(* Logix 5000 project; controller Turck_IOLink_All_Full_AOIs_V0_1 vendor 1 type 14 code 176 rev 32.11; software revision 32.00; part 4 of 7 *)
(* tags used below, declared in another part *)
   Port : INT;
   Common_Data : Turck_IOLink_Common_Data;   // Controller Tag of Process Data
   Units : SINT;   // Index 0x54 Subindex 1 - Change the Displayed Unit 0 = bar 1 = psi 2 = kPa 3 = MPa 4-14 = See Manual
   Rotate_Display : SINT;   // Index 0x5B - Subindex 1 - Display Rotation 0 = 0degrees 1 = 180 degrees
   Error : BOOL;
   Done : DINT;
   Error_DINT : DINT;
   Pending : DINT;
   Pending_or_Active : DINT;
   Units_Prev : SINT;
   StartupDone : BOOL;
   Active : DINT;
   Read_ONS : DINT;
   MyTicketNum : INT[32];
   Write : DINT;
   Write_ONS : DINT;
   WriteRequest : DINT;
   DoneCount : DINT;
   Status : DINT;
   ErrorCount : DINT;
   ReadRequest : DINT;
   Rotate_Display_Prev : SINT;
   Process_Data_Profile : SINT;
   Max_Pressure_Recorded_Raw : INT;
   Every_Min_Poll_TON : TIMER;
   Min_Recorded_Pressure_Raw : INT;
(* Turck_PS510_10V_Full, continued *)

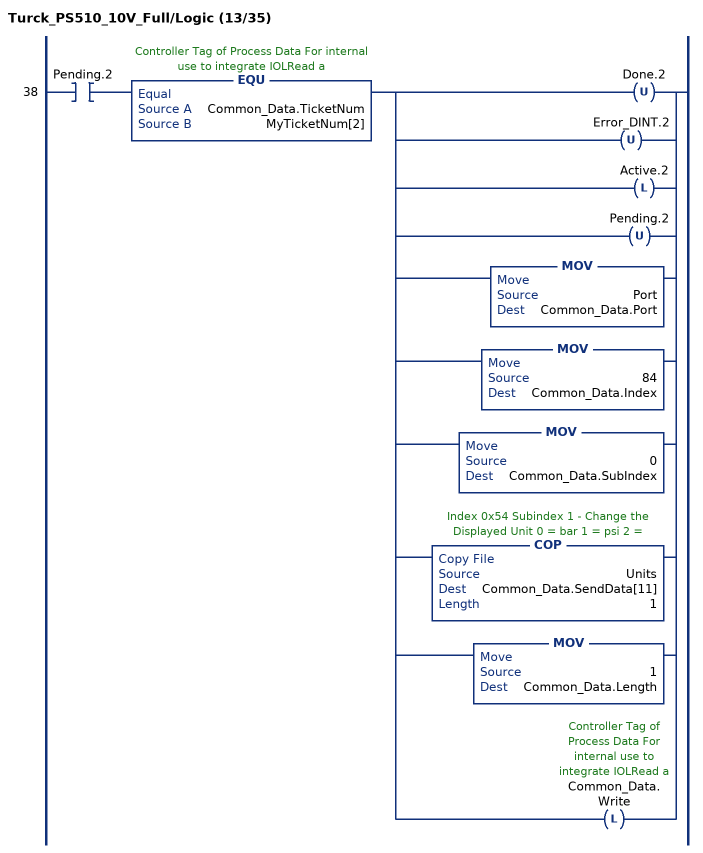
   [picture p75: Turck_PS510_10V_Full/Logic rungs 38-38]
   38: XIC(Pending.2)EQU(Common_Data.TicketNum,MyTicketNum[2])[OTU(Done.2) ,OTU(Error_DINT.2) ,OTL(Active.2) ,OTU(Pending.2) ,MOV(Port,Common_Data.Port) ,MOV(84,Common_Data.Index) ,MOV(0,Common_Data.SubIndex) ,COP(Units,Common_Data.SendData[11],1) ,MOV(1,Common_Data.Length) ,OTL(Common_Data.Write) ];
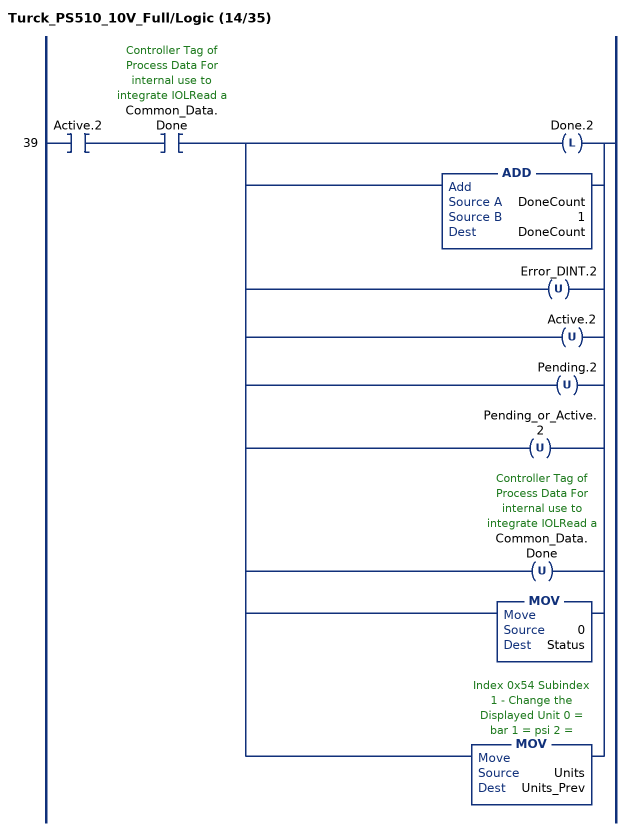
   39: XIC(Active.2)XIC(Common_Data.Done)[OTL(Done.2) ,ADD(DoneCount,1,DoneCount) ,OTU(Error_DINT.2) ,OTU(Active.2) ,OTU(Pending.2) ,OTU(Pending_or_Active.2) ,OTU(Common_Data.Done) ,MOV(0,Status) ,MOV(Units,Units_Prev) ];
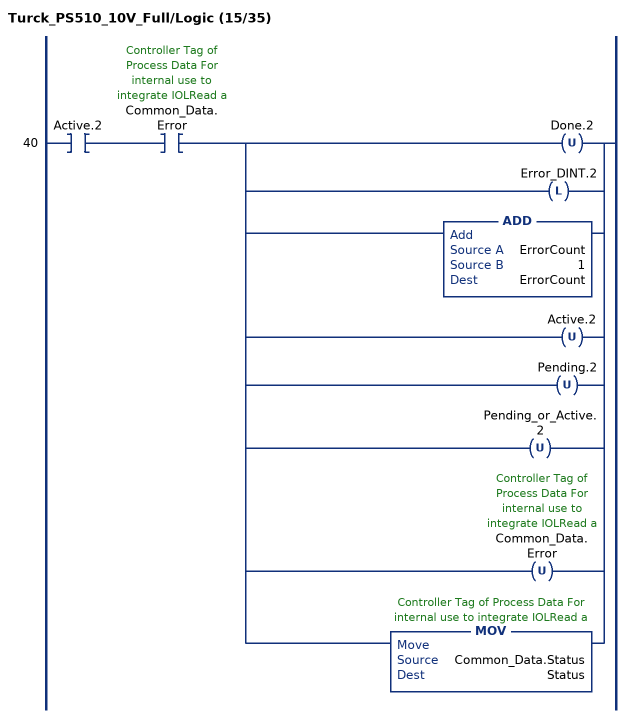
   40: XIC(Active.2)XIC(Common_Data.Error)[OTU(Done.2) ,OTL(Error_DINT.2) ,ADD(ErrorCount,1,ErrorCount) ,OTU(Active.2) ,OTU(Pending.2) ,OTU(Pending_or_Active.2) ,OTU(Common_Data.Error) ,MOV(Common_Data.Status,Status) ];
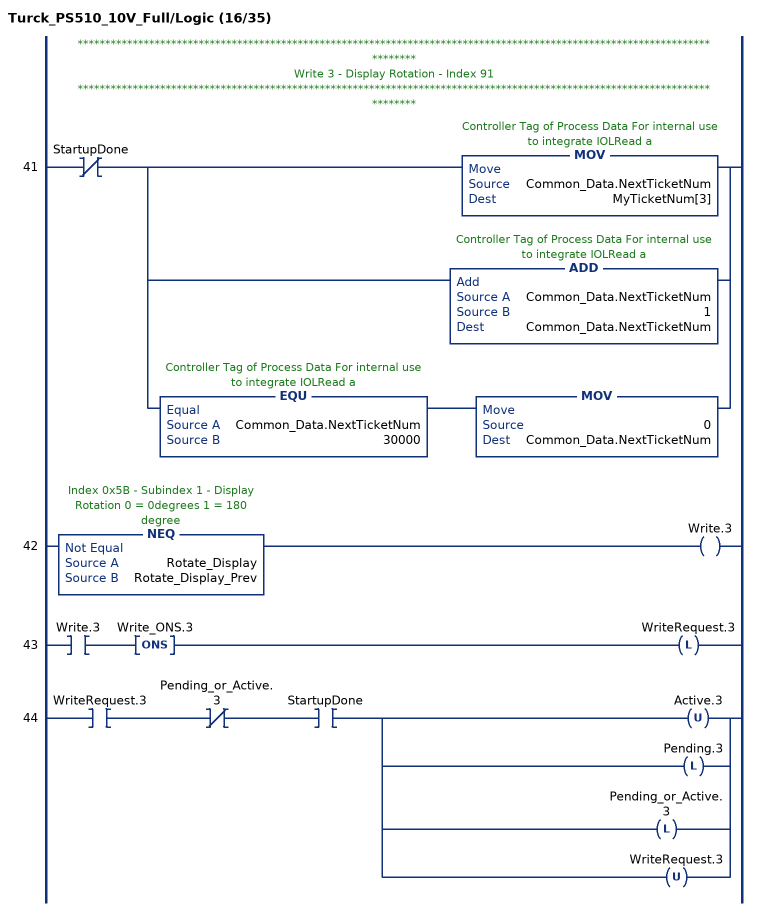
   // ***************************************************************************************************************************
   // Write 3 - Display Rotation - Index 91
   // ***************************************************************************************************************************
   41: XIO(StartupDone)[MOV(Common_Data.NextTicketNum,MyTicketNum[3]) ,ADD(Common_Data.NextTicketNum,1,Common_Data.NextTicketNum) ,EQU(Common_Data.NextTicketNum,30000) MOV(0,Common_Data.NextTicketNum) ];
   42: NEQ(Rotate_Display,Rotate_Display_Prev)OTE(Write.3);
   43: XIC(Write.3)ONS(Write_ONS.3)OTL(WriteRequest.3);
   44: XIC(WriteRequest.3)XIO(Pending_or_Active.3)XIC(StartupDone)[OTU(Active.3) ,OTL(Pending.3) ,OTL(Pending_or_Active.3) ,OTU(WriteRequest.3) ];
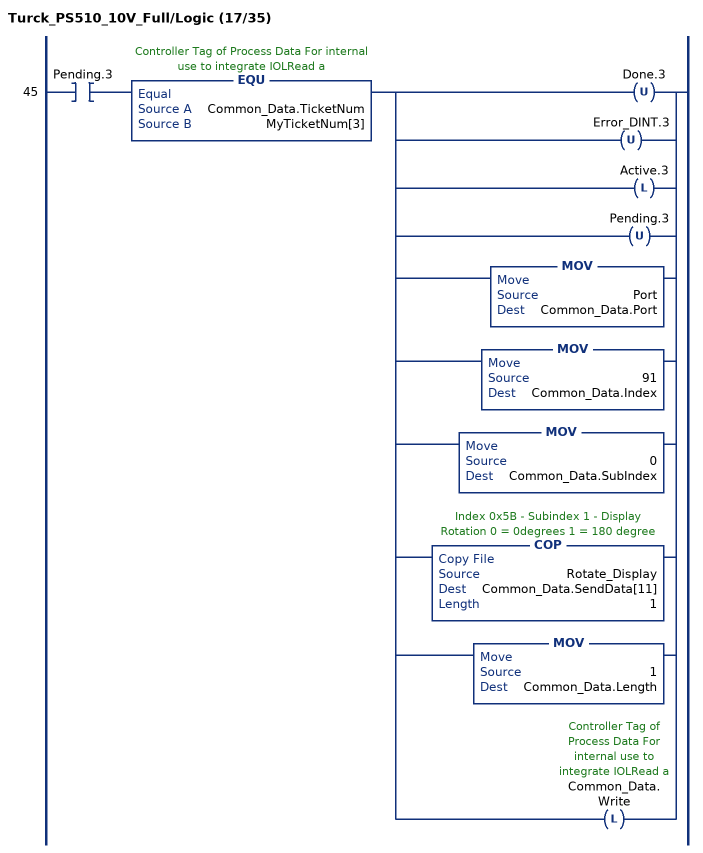
   45: XIC(Pending.3)EQU(Common_Data.TicketNum,MyTicketNum[3])[OTU(Done.3) ,OTU(Error_DINT.3) ,OTL(Active.3) ,OTU(Pending.3) ,MOV(Port,Common_Data.Port) ,MOV(91,Common_Data.Index) ,MOV(0,Common_Data.SubIndex) ,COP(Rotate_Display,Common_Data.SendData[11],1) ,MOV(1,Common_Data.Length) ,OTL(Common_Data.Write) ];
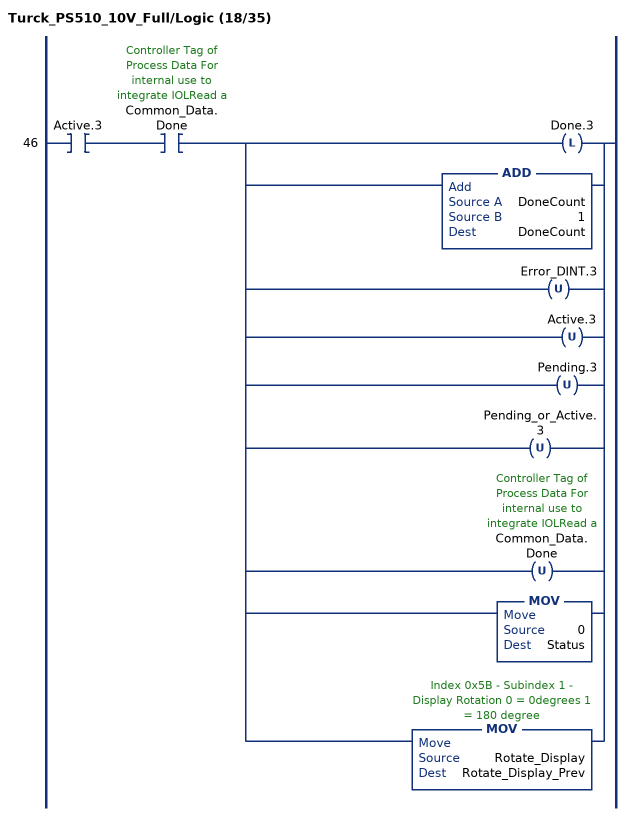
   46: XIC(Active.3)XIC(Common_Data.Done)[OTL(Done.3) ,ADD(DoneCount,1,DoneCount) ,OTU(Error_DINT.3) ,OTU(Active.3) ,OTU(Pending.3) ,OTU(Pending_or_Active.3) ,OTU(Common_Data.Done) ,MOV(0,Status) ,MOV(Rotate_Display,Rotate_Display_Prev) ];
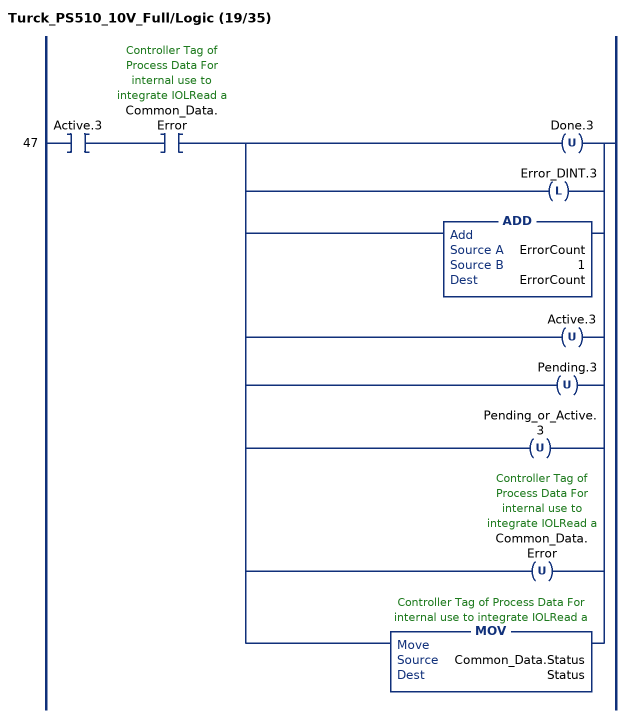
   47: XIC(Active.3)XIC(Common_Data.Error)[OTU(Done.3) ,OTL(Error_DINT.3) ,ADD(ErrorCount,1,ErrorCount) ,OTU(Active.3) ,OTU(Pending.3) ,OTU(Pending_or_Active.3) ,OTU(Common_Data.Error) ,MOV(Common_Data.Status,Status) ];
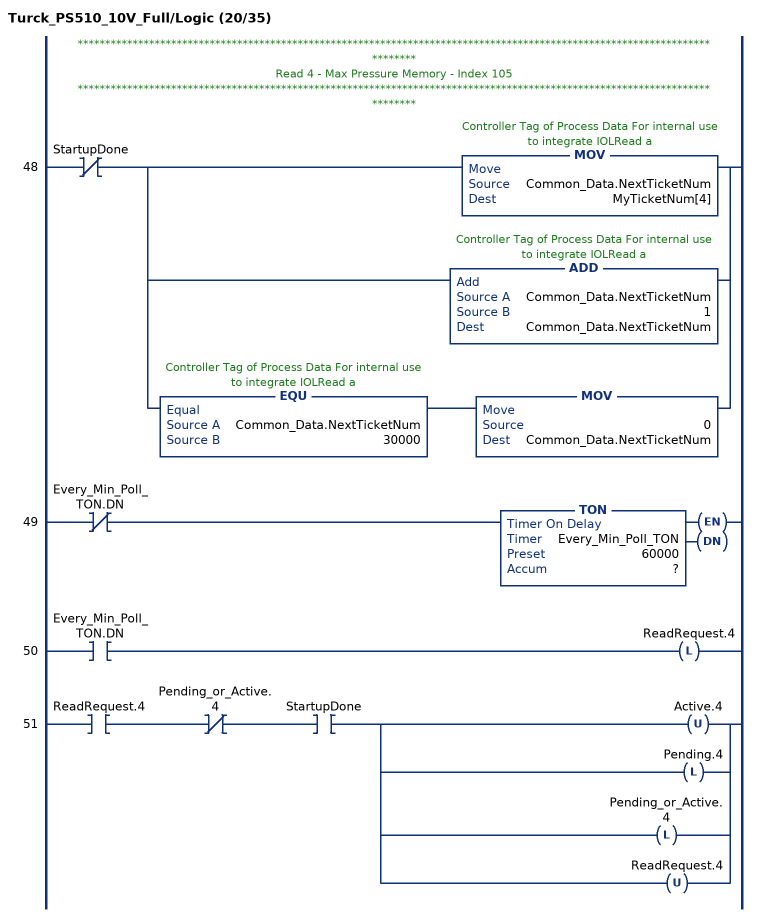
   // ***************************************************************************************************************************
   // Read 4 - Max Pressure Memory - Index 105
   // ***************************************************************************************************************************
   48: XIO(StartupDone)[MOV(Common_Data.NextTicketNum,MyTicketNum[4]) ,ADD(Common_Data.NextTicketNum,1,Common_Data.NextTicketNum) ,EQU(Common_Data.NextTicketNum,30000) MOV(0,Common_Data.NextTicketNum) ];
   49: XIO(Every_Min_Poll_TON.DN)TON(Every_Min_Poll_TON,?,?);
   50: XIC(Every_Min_Poll_TON.DN)OTL(ReadRequest.4);
   51: XIC(ReadRequest.4)XIO(Pending_or_Active.4)XIC(StartupDone)[OTU(Active.4) ,OTL(Pending.4) ,OTL(Pending_or_Active.4) ,OTU(ReadRequest.4) ];
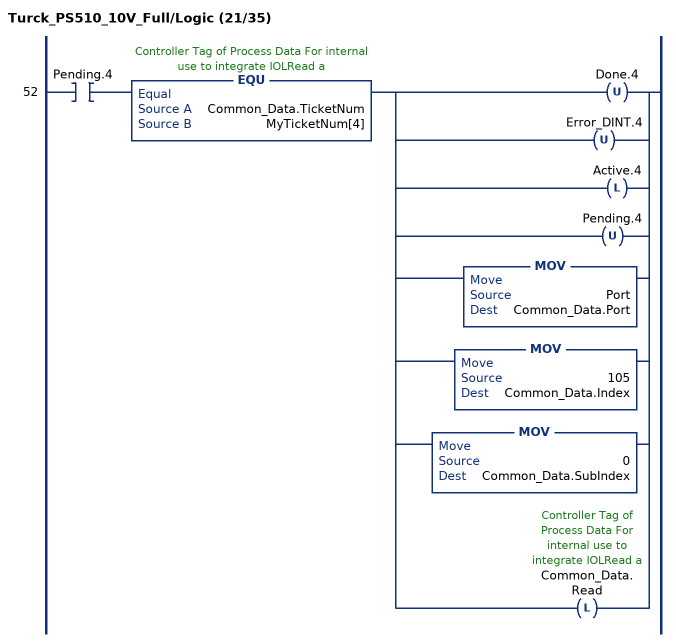
   52: XIC(Pending.4)EQU(Common_Data.TicketNum,MyTicketNum[4])[OTU(Done.4) ,OTU(Error_DINT.4) ,OTL(Active.4) ,OTU(Pending.4) ,MOV(Port,Common_Data.Port) ,MOV(105,Common_Data.Index) ,MOV(0,Common_Data.SubIndex) ,OTL(Common_Data.Read) ];
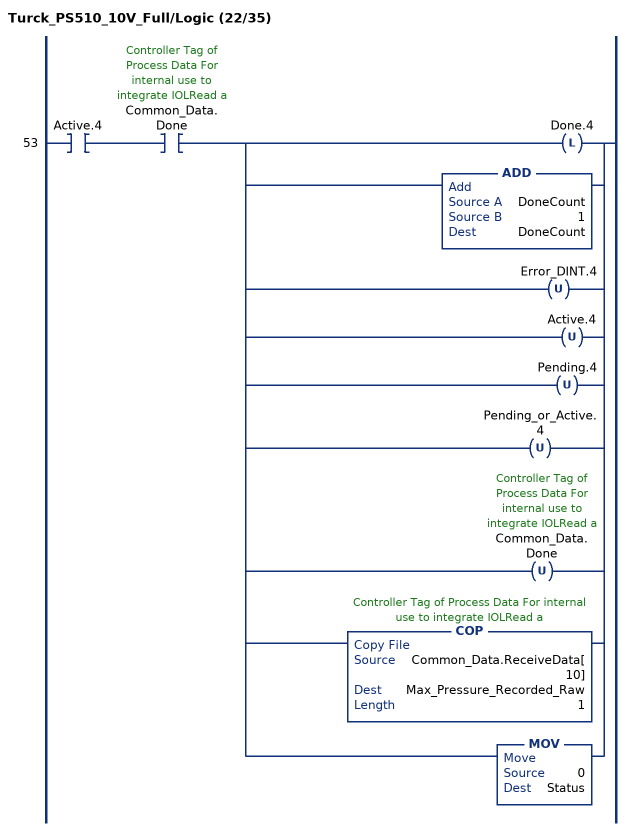
   53: XIC(Active.4)XIC(Common_Data.Done)[OTL(Done.4) ,ADD(DoneCount,1,DoneCount) ,OTU(Error_DINT.4) ,OTU(Active.4) ,OTU(Pending.4) ,OTU(Pending_or_Active.4) ,OTU(Common_Data.Done) ,COP(Common_Data.ReceiveData[10],Max_Pressure_Recorded_Raw,1) ,MOV(0,Status) ];
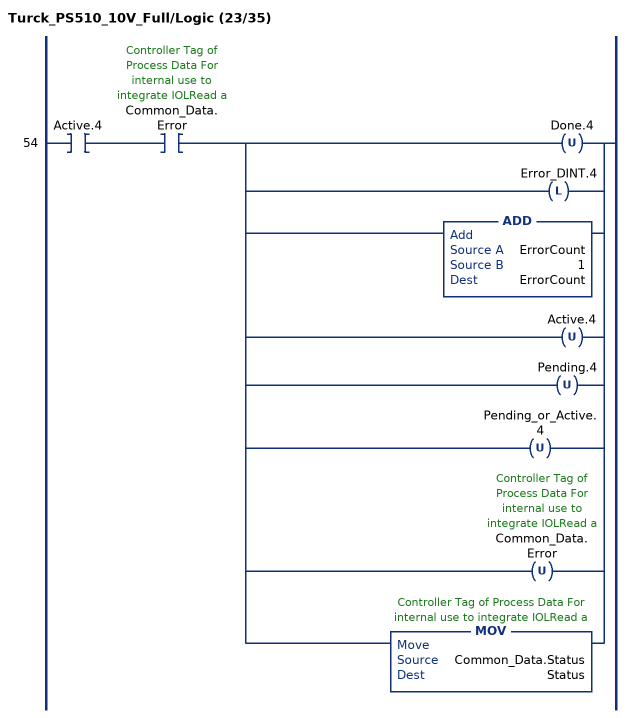
   54: XIC(Active.4)XIC(Common_Data.Error)[OTU(Done.4) ,OTL(Error_DINT.4) ,ADD(ErrorCount,1,ErrorCount) ,OTU(Active.4) ,OTU(Pending.4) ,OTU(Pending_or_Active.4) ,OTU(Common_Data.Error) ,MOV(Common_Data.Status,Status) ];
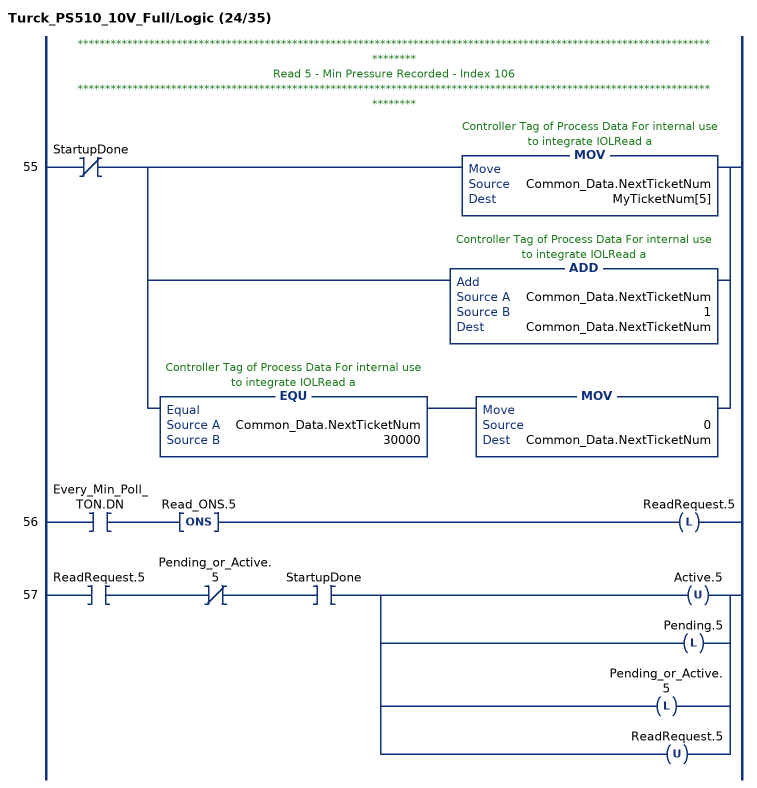
   // ***************************************************************************************************************************
   // Read 5 - Min Pressure Recorded - Index 106
   // ***************************************************************************************************************************
   55: XIO(StartupDone)[MOV(Common_Data.NextTicketNum,MyTicketNum[5]) ,ADD(Common_Data.NextTicketNum,1,Common_Data.NextTicketNum) ,EQU(Common_Data.NextTicketNum,30000) MOV(0,Common_Data.NextTicketNum) ];
   56: XIC(Every_Min_Poll_TON.DN)ONS(Read_ONS.5)OTL(ReadRequest.5);
   57: XIC(ReadRequest.5)XIO(Pending_or_Active.5)XIC(StartupDone)[OTU(Active.5) ,OTL(Pending.5) ,OTL(Pending_or_Active.5) ,OTU(ReadRequest.5) ];
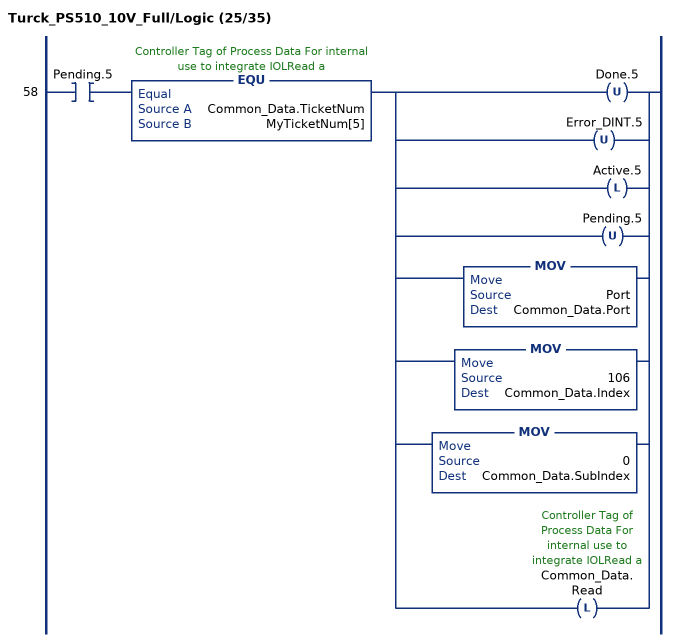
   58: XIC(Pending.5)EQU(Common_Data.TicketNum,MyTicketNum[5])[OTU(Done.5) ,OTU(Error_DINT.5) ,OTL(Active.5) ,OTU(Pending.5) ,MOV(Port,Common_Data.Port) ,MOV(106,Common_Data.Index) ,MOV(0,Common_Data.SubIndex) ,OTL(Common_Data.Read) ];
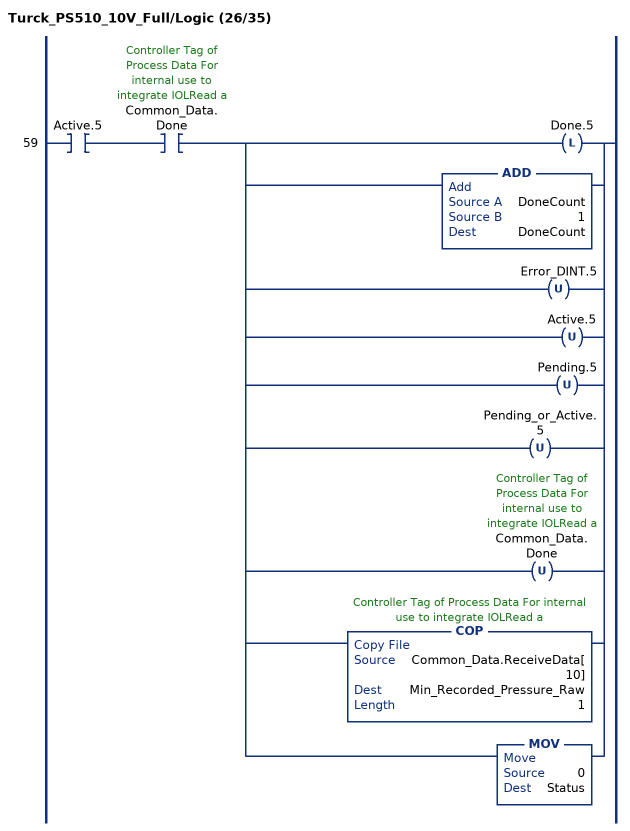
   59: XIC(Active.5)XIC(Common_Data.Done)[OTL(Done.5) ,ADD(DoneCount,1,DoneCount) ,OTU(Error_DINT.5) ,OTU(Active.5) ,OTU(Pending.5) ,OTU(Pending_or_Active.5) ,OTU(Common_Data.Done) ,COP(Common_Data.ReceiveData[10],Min_Recorded_Pressure_Raw,1) ,MOV(0,Status) ];
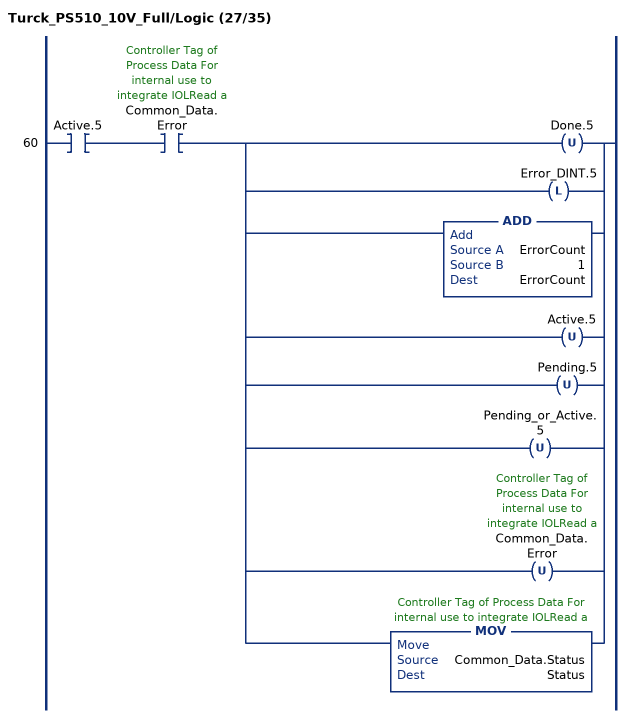
   60: XIC(Active.5)XIC(Common_Data.Error)[OTU(Done.5) ,OTL(Error_DINT.5) ,ADD(ErrorCount,1,ErrorCount) ,OTU(Active.5) ,OTU(Pending.5) ,OTU(Pending_or_Active.5) ,OTU(Common_Data.Error) ,MOV(Common_Data.Status,Status) ];
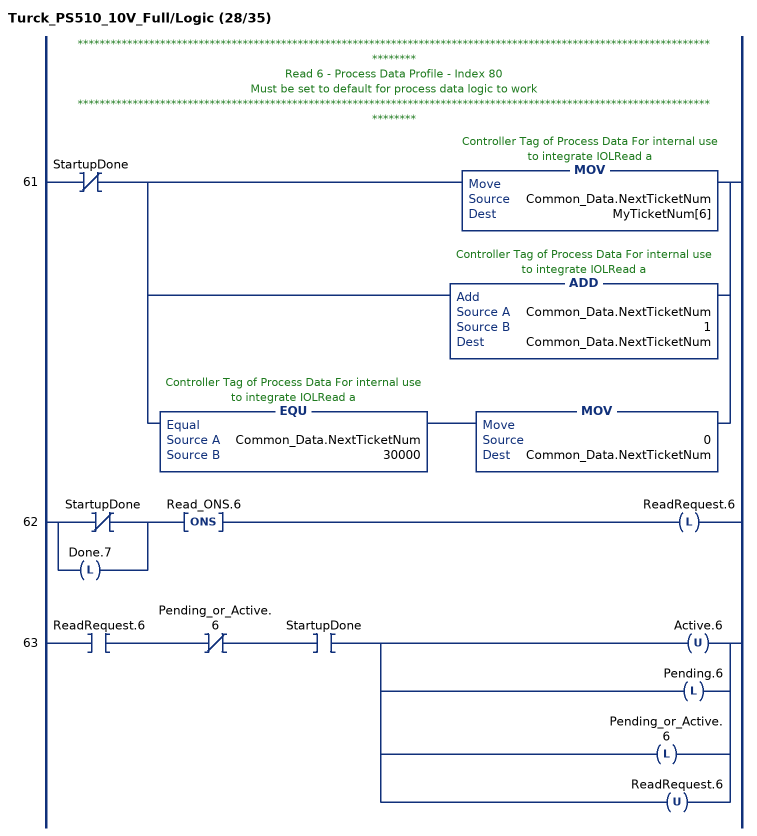
   // ***************************************************************************************************************************
   // Read 6 - Process Data Profile - Index 80
   // Must be set to default for process data logic to work
   // ***************************************************************************************************************************
   61: XIO(StartupDone)[MOV(Common_Data.NextTicketNum,MyTicketNum[6]) ,ADD(Common_Data.NextTicketNum,1,Common_Data.NextTicketNum) ,EQU(Common_Data.NextTicketNum,30000) MOV(0,Common_Data.NextTicketNum) ];
   62: [XIO(StartupDone) ,OTL(Done.7) ]ONS(Read_ONS.6)OTL(ReadRequest.6);
   63: XIC(ReadRequest.6)XIO(Pending_or_Active.6)XIC(StartupDone)[OTU(Active.6) ,OTL(Pending.6) ,OTL(Pending_or_Active.6) ,OTU(ReadRequest.6) ];
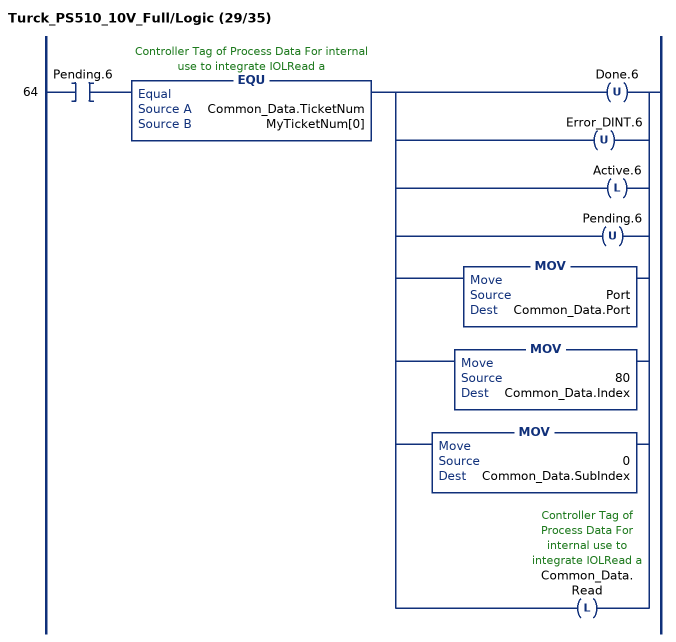
   64: XIC(Pending.6)EQU(Common_Data.TicketNum,MyTicketNum[0])[OTU(Done.6) ,OTU(Error_DINT.6) ,OTL(Active.6) ,OTU(Pending.6) ,MOV(Port,Common_Data.Port) ,MOV(80,Common_Data.Index) ,MOV(0,Common_Data.SubIndex) ,OTL(Common_Data.Read) ];
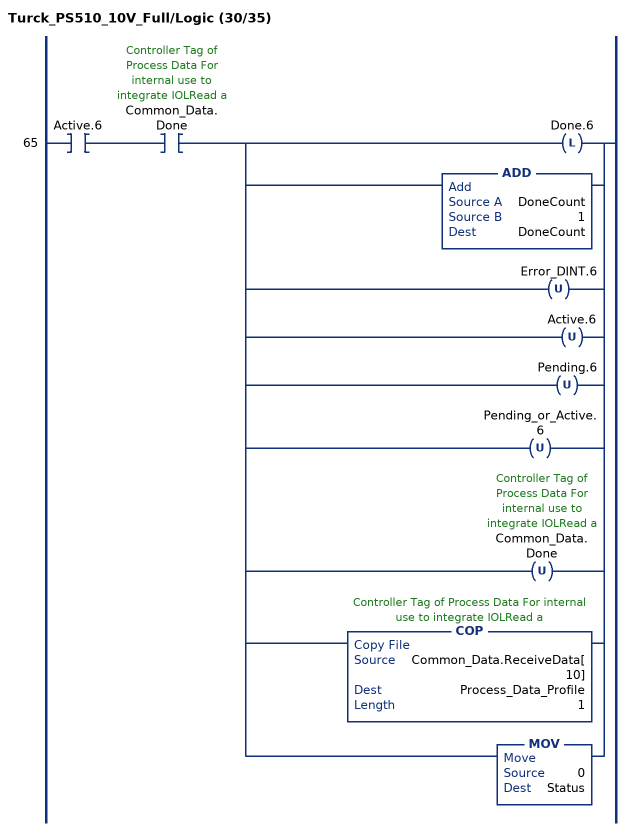
   65: XIC(Active.6)XIC(Common_Data.Done)[OTL(Done.6) ,ADD(DoneCount,1,DoneCount) ,OTU(Error_DINT.6) ,OTU(Active.6) ,OTU(Pending.6) ,OTU(Pending_or_Active.6) ,OTU(Common_Data.Done) ,COP(Common_Data.ReceiveData[10],Process_Data_Profile,1) ,MOV(0,Status) ];
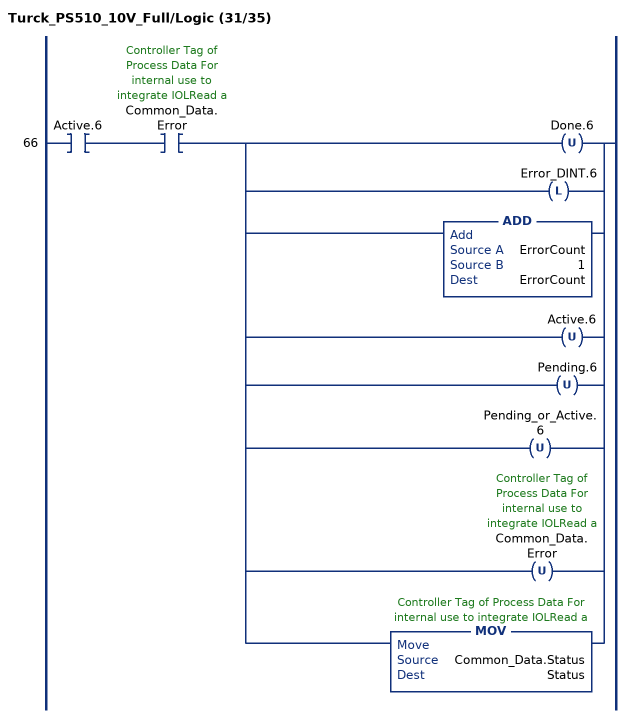
   66: XIC(Active.6)XIC(Common_Data.Error)[OTU(Done.6) ,OTL(Error_DINT.6) ,ADD(ErrorCount,1,ErrorCount) ,OTU(Active.6) ,OTU(Pending.6) ,OTU(Pending_or_Active.6) ,OTU(Common_Data.Error) ,MOV(Common_Data.Status,Status) ];
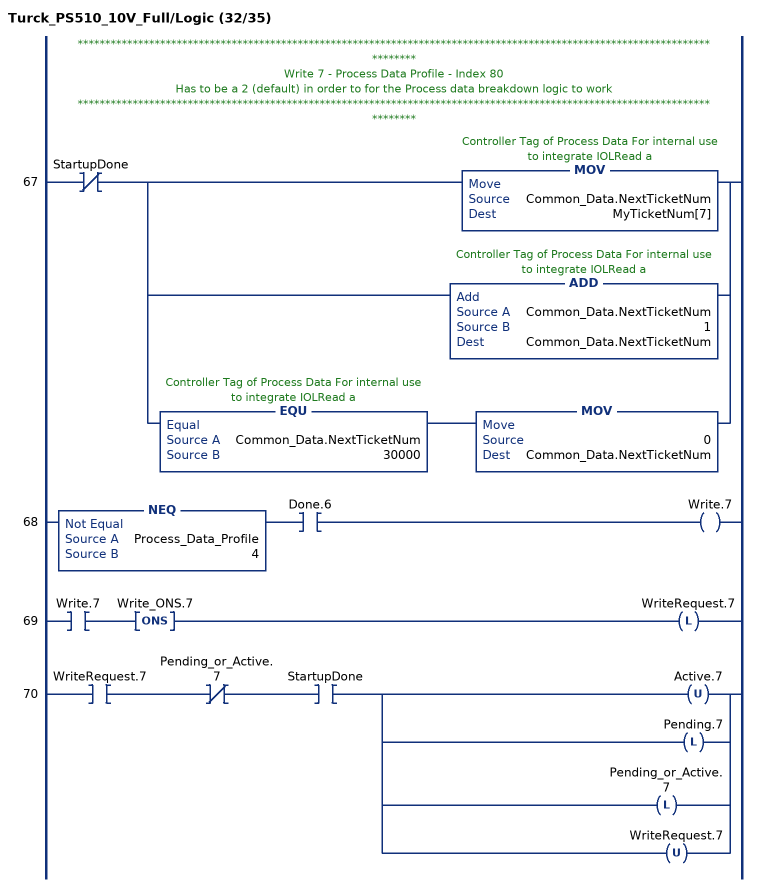
   // ***************************************************************************************************************************
   // Write 7 - Process Data Profile - Index 80
   // Has to be a 2 (default) in order to for the Process data breakdown logic to work
   // ***************************************************************************************************************************
   67: XIO(StartupDone)[MOV(Common_Data.NextTicketNum,MyTicketNum[7]) ,ADD(Common_Data.NextTicketNum,1,Common_Data.NextTicketNum) ,EQU(Common_Data.NextTicketNum,30000) MOV(0,Common_Data.NextTicketNum) ];
   68: NEQ(Process_Data_Profile,4)XIC(Done.6)OTE(Write.7);
   69: XIC(Write.7)ONS(Write_ONS.7)OTL(WriteRequest.7);
   70: XIC(WriteRequest.7)XIO(Pending_or_Active.7)XIC(StartupDone)[OTU(Active.7) ,OTL(Pending.7) ,OTL(Pending_or_Active.7) ,OTU(WriteRequest.7) ];
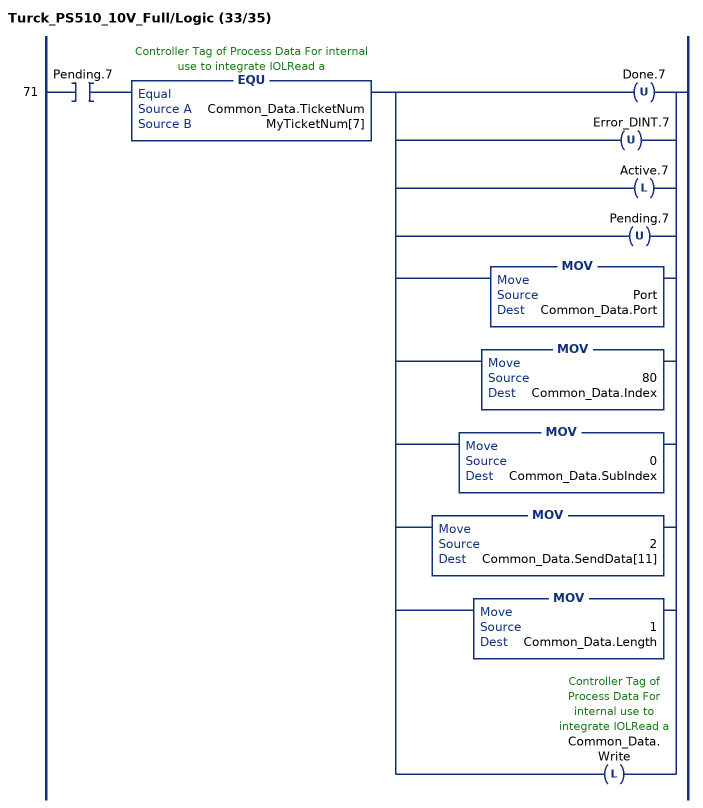
   71: XIC(Pending.7)EQU(Common_Data.TicketNum,MyTicketNum[7])[OTU(Done.7) ,OTU(Error_DINT.7) ,OTL(Active.7) ,OTU(Pending.7) ,MOV(Port,Common_Data.Port) ,MOV(80,Common_Data.Index) ,MOV(0,Common_Data.SubIndex) ,MOV(2,Common_Data.SendData[11]) ,MOV(1,Common_Data.Length) ,OTL(Common_Data.Write) ];
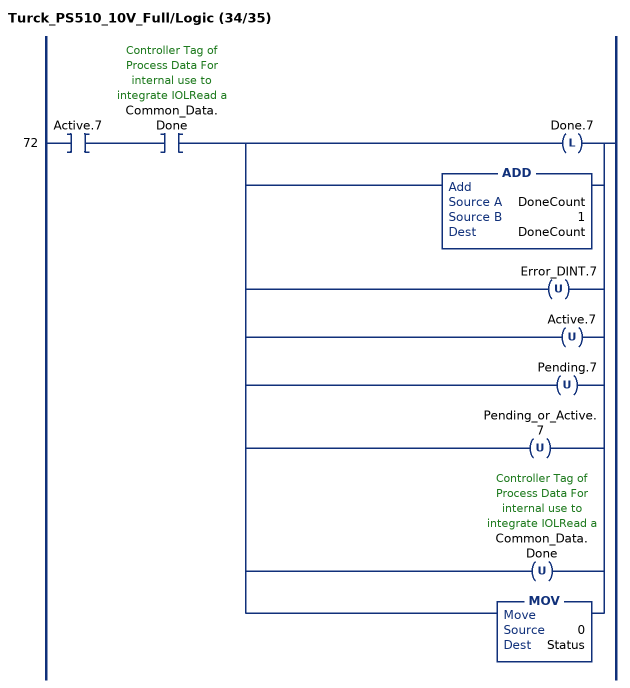
   72: XIC(Active.7)XIC(Common_Data.Done)[OTL(Done.7) ,ADD(DoneCount,1,DoneCount) ,OTU(Error_DINT.7) ,OTU(Active.7) ,OTU(Pending.7) ,OTU(Pending_or_Active.7) ,OTU(Common_Data.Done) ,MOV(0,Status) ];
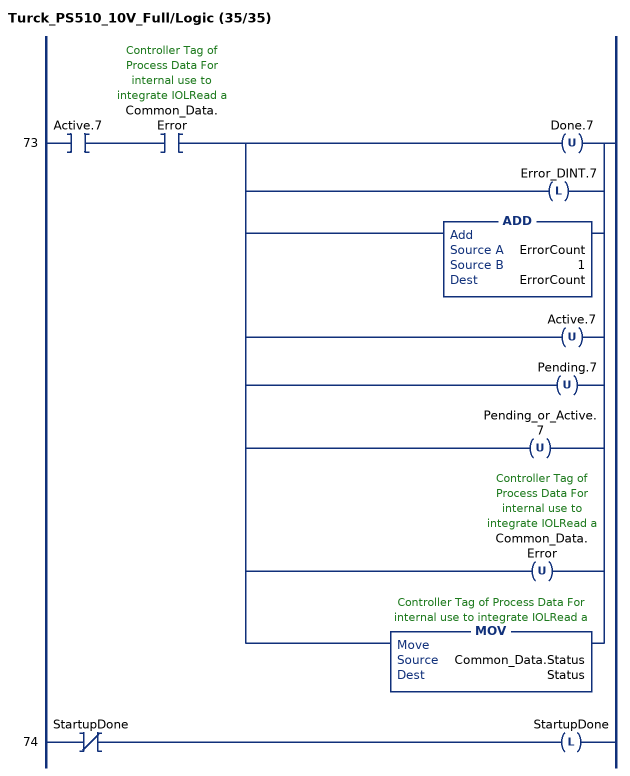
   73: XIC(Active.7)XIC(Common_Data.Error)[OTU(Done.7) ,OTL(Error_DINT.7) ,ADD(ErrorCount,1,ErrorCount) ,OTU(Active.7) ,OTU(Pending.7) ,OTU(Pending_or_Active.7) ,OTU(Common_Data.Error) ,MOV(Common_Data.Status,Status) ];
   74: XIO(StartupDone)OTL(StartupDone);
END_ROUTINE
